(*

short summary
=============

.. <legal notes>

legal notes
=================
| SPDX-FileCopyrightText: © 2023 ekvip automation GmbH <info@ekvip.de>
| SPDX-License-Identifier: Apache-2.0
| For details check: Apache-2.0_

.. _Apache-2.0: https://www.apache.org/licenses/LICENSE-2.0

.. </legal notes>

*)

{warning 'header is generated please add your documentation'}
TYPE AnyTestString :
STRUCT
	wstringToTest	:WSTRING(300);
	stringToTest	:STRING(600);
END_STRUCT
END_TYPE

(* stored: Version 1.1.0.1, ProductVersion 3.1.4024.12
   DUT AnyTestString: Id {5d720692-c272-4d7c-9d5e-9540222bef37} *)
